// TIA Portal V17 export
FUNCTION "FC_VFD_CommFault" : Void   // FC, LAD
{ S7_Optimized_Access := 'TRUE' }
BEGIN
END_FUNCTION
